// TIA Portal V20 export
TYPE "typeSequenceControlNodeHomeCheck"
// stored: Namespace Unit1.Em9
   STRUCT
      liftDownLightUpPartNoDetect : Bool;
      liftDownLightUpPartDetect : Bool;
      liftDownLightDownPartDetect : Bool;
      liftUpLightUp : Bool;
   END_STRUCT;
END_TYPE
